FUNCTION_BLOCK FB_FieldCodecInt64 EXTENDS FB_FieldCodec
VAR_INPUT
END_VAR
VAR_OUTPUT
END_VAR
VAR
    nValue : ULINT;
END_VAR

METHOD CalculatePackedDataSize : HRESULT
VAR_INPUT CONSTANT
	anyFirstElem	: T_Any;
	nLength	        : UDINT;        // items to write
END_VAR
VAR_OUTPUT
    nPackedDataSize : UDINT;
END_VAR
VAR
    anyItem         : T_ANY;
    i               : UDINT;
    nValue          : LINT;
END_VAR
anyItem := anyFirstElem;

IF nLength < 1 THEN
    nPackedDataSize := 0;
    RETURN;
END_IF

FOR i := 0  TO nLength - 1 DO
    anyItem.pValue := anyFirstElem.pValue + (i * TO_UDINT(anyFirstElem.diSize)); 
    nValue := PLINT_TO_LINT(anyItem.pValue);
    nPackedDataSize := nPackedDataSize + F_ComputeInt64Size(nValue);
END_FOR
END_METHOD

METHOD IsPackedRepeatedField : BOOL
VAR_INPUT
	nTag	: UDINT;
END_VAR
IsPackedRepeatedField := F_IsPackedRepeatedField(nTag);
END_METHOD


METHOD ValueReader : HRESULT
VAR_IN_OUT      
    stCtx : ST_ParseContext;
END_VAR
VAR_OUTPUT
	anyOut	: T_Any;
END_VAR

ValueReader := F_ParseRawVarint64(stCtx, nValue);
anyOut := F_ToAnyType(anyArg:= nValue);
END_METHOD

METHOD ValueWriter : HRESULT
VAR_IN_OUT
    stCtx  : ST_WriteContext;
END_VAR
VAR_INPUT
    anyIn : T_ANY;
END_VAR
VAR
    nValue  : LINT;
END_VAR

nValue := PLINT_TO_LINT(anyIn.pValue);
ValueWriter := F_WriteInt64(stCtx, nValue);
END_METHOD

END_FUNCTION_BLOCK

(* stored: Version 1.1.0.1
   POU FB_FieldCodecInt64: Id {fb13e9c5-307a-437d-b4d8-44df2b27263e}, SpecialFunc None
   Method CalculatePackedDataSize: Id {aab6e214-2d04-4c47-8787-60d46a9f570e}
   Method IsPackedRepeatedField: Id {5d2ced4d-5bc7-40e4-ba18-9751afd814db}
   Method ValueReader: Id {82106cf7-1545-4b64-9960-92a4b19900dc}
   Method ValueWriter: Id {743d62ea-3845-45ce-b389-9a69a8933713} *)
